(*			
	RAFALOS
	Rafał Osajda		19.09.2025		TC 4024.66
	FB Bazowy dla wszystkich elementów złożonych
*)
FUNCTION_BLOCK FB_BaseGroupElement EXTENDS FB_BaseControlElement IMPLEMENTS ITF_BaseGroupElement, ITF_BaseGroupElement_HMI_Connector
VAR
	arrControlElement			: ARRAY [1..GVL_BaseConstans.MAX_ITEM_PER_ELEMENT] OF ITF_BaseControlElement;
	uiNumberOfControlElement	: UINT;
END_VAR

METHOD PROTECTED AddControlElement : BOOL
VAR_INPUT
	itfControlElement		: ITF_BaseControlElement;
END_VAR
IF (THIS^.uiNumberOfControlElement + 1 <= GVL_BaseConstans.MAX_ITEM_PER_ELEMENT) THEN
	THIS^.uiNumberOfControlElement		:= THIS^.uiNumberOfControlElement + 1;
	THIS^.arrControlElement [THIS^.uiNumberOfControlElement]	:= itfControlElement;
	AddControlElement			:= TRUE;
ELSE
	;//zwrocenie zbyt dużo komponentow
END_IF
END_METHOD

METHOD FB_init : BOOL
VAR_INPUT
	bInitRetains : BOOL; // if TRUE, the retain variables are initialized (warm start / cold start)
	bInCopyCode : BOOL;  // if TRUE, the instance afterwards gets moved into the copy code (online change)
END_VAR
THIS^.stIdentifier.eType			:= E_BaseElementType.eGroup;
END_METHOD

METHOD PUBLIC FirstCycle : BOOL
VAR_INPUT
END_VAR
VAR
	bResult			: bool;
	iI				: INT;
END_VAR
bResult				:= SUPER^.FirstCycle ();

FOR iI := 1 TO TO_INT (THIS^.uiNumberOfControlElement) DO
	bResult			:= bResult AND THIS^.arrControlElement [iI].FirstCycle ();
END_FOR

FirstCycle			:= bResult;
END_METHOD

METHOD PUBLIC IsValidCommonData : BOOL
VAR_INPUT
END_VAR

VAR
	bResult: BOOL;
	iI: INT;
END_VAR
bResult						:= SUPER^.IsValidCommonData ();

FOR iI := 1 TO TO_INT (THIS^.uiNumberOfControlElement) DO
	bResult					:= bResult AND THIS^.arrControlElement [iI].IsValidCommonData ();
END_FOR

IsValidCommonData			:= bResult;
END_METHOD

METHOD PUBLIC LinkCommonData : BOOL
VAR_INPUT
	stCommonData				: REFERENCE TO ST_BaseCommonData;
END_VAR
VAR
	bResult						: BOOL;
	iI: INT;
END_VAR
bResult							:= SUPER^.LinkCommonData (stCommonData := stCommonData);

FOR iI := 1 TO TO_INT (THIS^.uiNumberOfControlElement) DO
	bResult := bResult AND THIS^.arrControlElement [iI].LinkCommonData (stCommonData := stCommonData);
END_FOR

LinkCommonData					:= bResult;
END_METHOD

(*			
	EVERDE sp. z o.o.
	Rafał Osajda		03.10.2025		TC 4024.66
	nadawanie unikalnych ID dla zdarzeń
*)
METHOD PUBLIC SetEventsIDs : UINT
VAR_INPUT
	uiNewID		: UINT;
END_VAR
VAR
	iI			: INT;
	uiLastID	: UINT;
END_VAR
uiLastID		:= SUPER^.SetEventsIDs (uiNewID	:= uiNewID);

FOR iI := 1 TO TO_INT (THIS^.uiNumberOfControlElement) DO 
	uiLastID			:= THIS^.arrControlElement [iI].SetEventsIDs (uiNewID	:= uiLastID);
END_FOR
SetEventsIDs				:= uiLastID;
END_METHOD

END_FUNCTION_BLOCK

(* stored: Version 1.1.0.1
   POU FB_BaseGroupElement: Id {1f8518b0-2e03-0c13-2a4a-ffc3b6f9b887}, SpecialFunc None
   Folder Events: Id {20f6f417-5dd7-052c-022d-8978faa14be3}
   Folder WiazanieZmiennych: Id {2b50b030-a9ec-06ce-1ddf-f0356b93fad0}
   Method AddControlElement: Id {175b37ba-638b-0727-26cf-573800512486}
   Method FB_init: Id {a18f7400-8689-05ae-3b31-59cab5e8ddb8}
   Method FirstCycle: Id {fede4491-2815-0c5d-25f3-a52cafaf5311}
   Method IsValidCommonData: Id {f68feac5-aff9-07a7-017f-3067903007ab}
   Method LinkCommonData: Id {163c9121-a3cf-0bfe-2517-ea6f42e3be4a}
   Method SetEventsIDs: Id {0185e120-5cb8-0dba-3756-ff856ef7df3c} *)
